% RSLogix 500 project FOUNTAIN.RSS, saved by version 8.30.00.16 %
PROJECT "UNTITLED"    % processor: MicroLogix 1000 %

PROGRAM FILES
  LAD 2 "MAIN_PROG"  26 rungs
  LAD 3 "COUNTER"  1 rungs
  LAD 4 "FLASHER"  1 rungs
  LAD 5 "STI_INT"  1 rungs
  LAD 6, 7, 8, 9, 10, 11, 12, 13, 14, 15, 16: only END

DATA FILES
  O0 OUTPUT  1 elements
  I1 INPUT  2 elements
  S2 STATUS  33 elements
  B3 BINARY  32 elements
  T4 TIMER  40 elements
  C5 COUNTER  32 elements
  R6 CONTROL  16 elements
  N7 INTEGER  105 elements

LADDER 2 "MAIN_PROG"
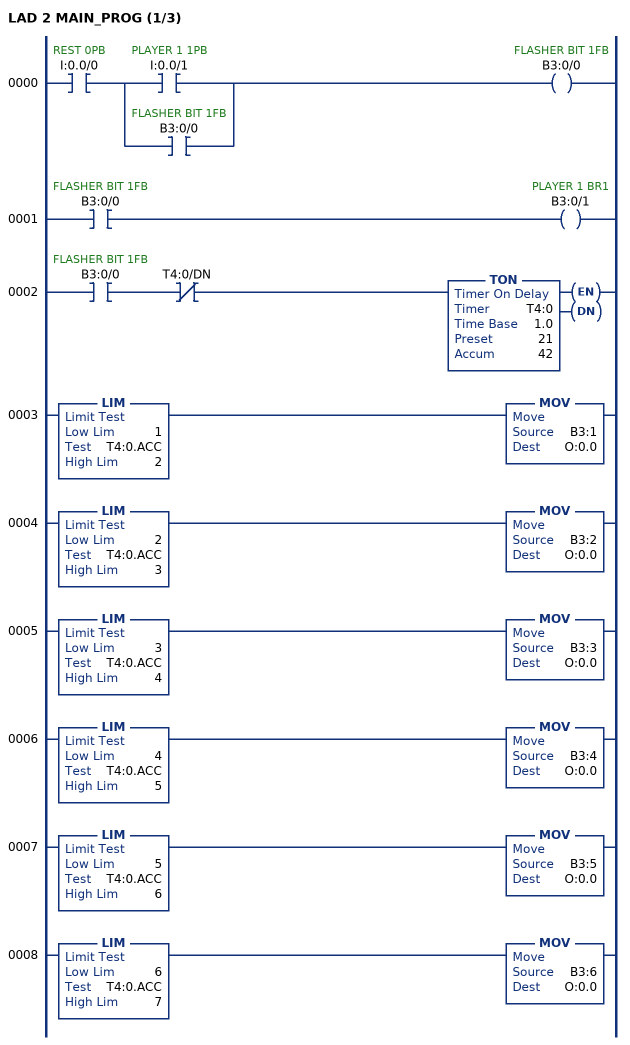
% Rung: 0 %
SOR XIC I:0.0/0 BST XIC I:0.0/1 NXB XIC B3:0/0 BND OTE B3:0/0 EOR
%   I:0.0/0  0PB  "REST" %
%   I:0.0/1  1PB  "PLAYER 1" %
%   B3:0/0  1FB  "FLASHER BIT" %
% Rung: 1 %
SOR XIC B3:0/0 OTE B3:0/1 EOR
%   B3:0/0  1FB  "FLASHER BIT" %
%   B3:0/1  BR1  "PLAYER 1" %
% Rung: 2 %
SOR XIC B3:0/0 XIO T4:0/DN TON T4:0 1.0 21 42 EOR
%   B3:0/0  1FB  "FLASHER BIT" %
% Rung: 3 %
SOR LIM 1 T4:0.ACC 2 MOV B3:1 O:0.0 EOR
% Rung: 4 %
SOR LIM 2 T4:0.ACC 3 MOV B3:2 O:0.0 EOR
% Rung: 5 %
SOR LIM 3 T4:0.ACC 4 MOV B3:3 O:0.0 EOR
% Rung: 6 %
SOR LIM 4 T4:0.ACC 5 MOV B3:4 O:0.0 EOR
% Rung: 7 %
SOR LIM 5 T4:0.ACC 6 MOV B3:5 O:0.0 EOR
% Rung: 8 %
SOR LIM 6 T4:0.ACC 7 MOV B3:6 O:0.0 EOR

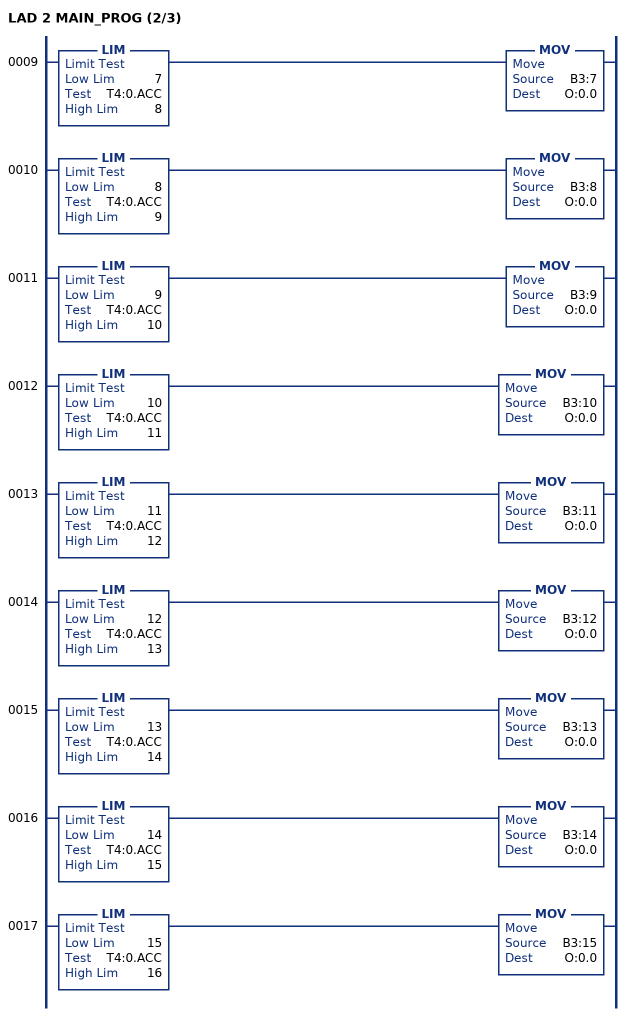
% Rung: 9 %
SOR LIM 7 T4:0.ACC 8 MOV B3:7 O:0.0 EOR
% Rung: 10 %
SOR LIM 8 T4:0.ACC 9 MOV B3:8 O:0.0 EOR
% Rung: 11 %
SOR LIM 9 T4:0.ACC 10 MOV B3:9 O:0.0 EOR
% Rung: 12 %
SOR LIM 10 T4:0.ACC 11 MOV B3:10 O:0.0 EOR
% Rung: 13 %
SOR LIM 11 T4:0.ACC 12 MOV B3:11 O:0.0 EOR
% Rung: 14 %
SOR LIM 12 T4:0.ACC 13 MOV B3:12 O:0.0 EOR
% Rung: 15 %
SOR LIM 13 T4:0.ACC 14 MOV B3:13 O:0.0 EOR
% Rung: 16 %
SOR LIM 14 T4:0.ACC 15 MOV B3:14 O:0.0 EOR
% Rung: 17 %
SOR LIM 15 T4:0.ACC 16 MOV B3:15 O:0.0 EOR

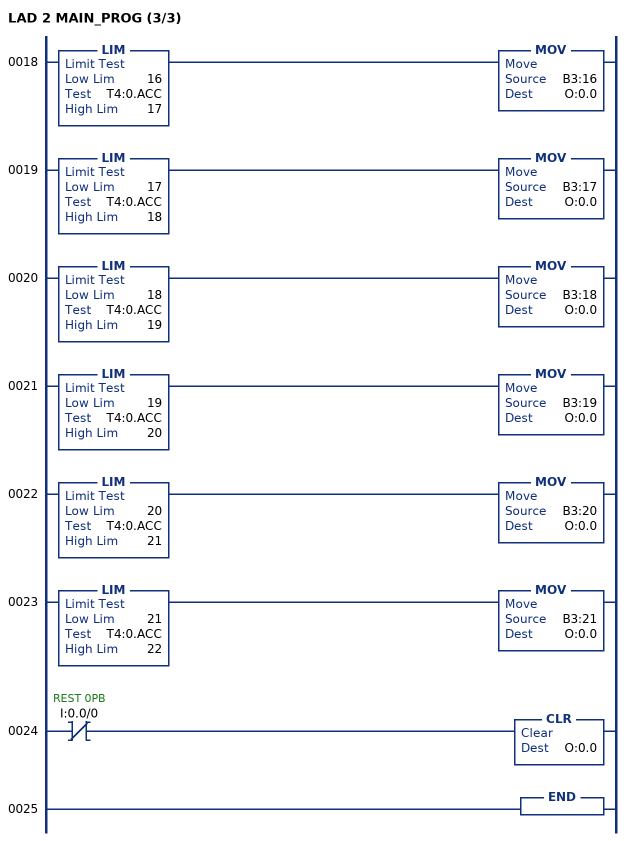
% Rung: 18 %
SOR LIM 16 T4:0.ACC 17 MOV B3:16 O:0.0 EOR
% Rung: 19 %
SOR LIM 17 T4:0.ACC 18 MOV B3:17 O:0.0 EOR
% Rung: 20 %
SOR LIM 18 T4:0.ACC 19 MOV B3:18 O:0.0 EOR
% Rung: 21 %
SOR LIM 19 T4:0.ACC 20 MOV B3:19 O:0.0 EOR
% Rung: 22 %
SOR LIM 20 T4:0.ACC 21 MOV B3:20 O:0.0 EOR
% Rung: 23 %
SOR LIM 21 T4:0.ACC 22 MOV B3:21 O:0.0 EOR
% Rung: 24 %
SOR XIO I:0.0/0 CLR O:0.0 EOR
%   I:0.0/0  0PB  "REST" %
% Rung: 25 %
SOR END EOR

OTHER DOCUMENTED ADDRESSES
  B3  
  B3:0/2  BR2  "PLAYER 2"
  B3:0/3  BR3  "PLAYER 3"
  B3:0/4  BT4  "PLAYER 1"
  B3:0/5  BT5  "PLAYER 2"
  B3:0/6  BT6  "PLAYER 3"
  B3:0/7  BT7  "PLAYER 1"
  B3:0/8  BT8  "PLAYER 2"
  B3:0/9  BT_9  "PLAYER 3"
  B30:0/1  1BT  "PLAYER 1"
  B30:0/2  BT2  "PLAYER 2"
  B30:0/3  BT3  "PLAYER 3"
  C5:0  1C  "FLASHER COUNTER"
  I:0.0/2  2PB  "PLAYER 2"
  I:0.0/3  3PB  "PLAYER 3"
  O:0.0/0  0LT  "PLAYER START"
  O:0.0/1  1TH  "PLAYER 1"
  O:0.0/2  2LT  "PLAYER 2"
  O:0.0/3  3LT  "PLAYER 3"
  O:0.0/4  RST  "REST"
  O:0.0/5  "RESET STOP"
  T4:1  2FTOF  "FLASHER OFF TIMER"
  T4:2  1FTON  "FLASHER ON TIMER"
  T4:2/DN  "FLASHER OFF TIMER"
  U:3  "FLASHER COUNTER"
  U:4  "FLASHER"

DATA TABLE (non-zero values as saved)
DATA B3
% B3:0 % 0X0003 0X0001 0X0002 0X0004 0X0008 0X0000 0X0008 0X0004 0X0002 0X0001
% B3:10 % 0X0000 0X000F 0X0009 0X0006 0X0009 0X0006 0X0009 0X0005 0X000A 0X0005
% B3:20 % 0X000A 0X0000 0X0000 0X0000 0X0000 0X0000 0X0000 0X0000 0X0000 0X0000
DATA T4
% .PRE .ACC %
% T4:0 % 21 42
